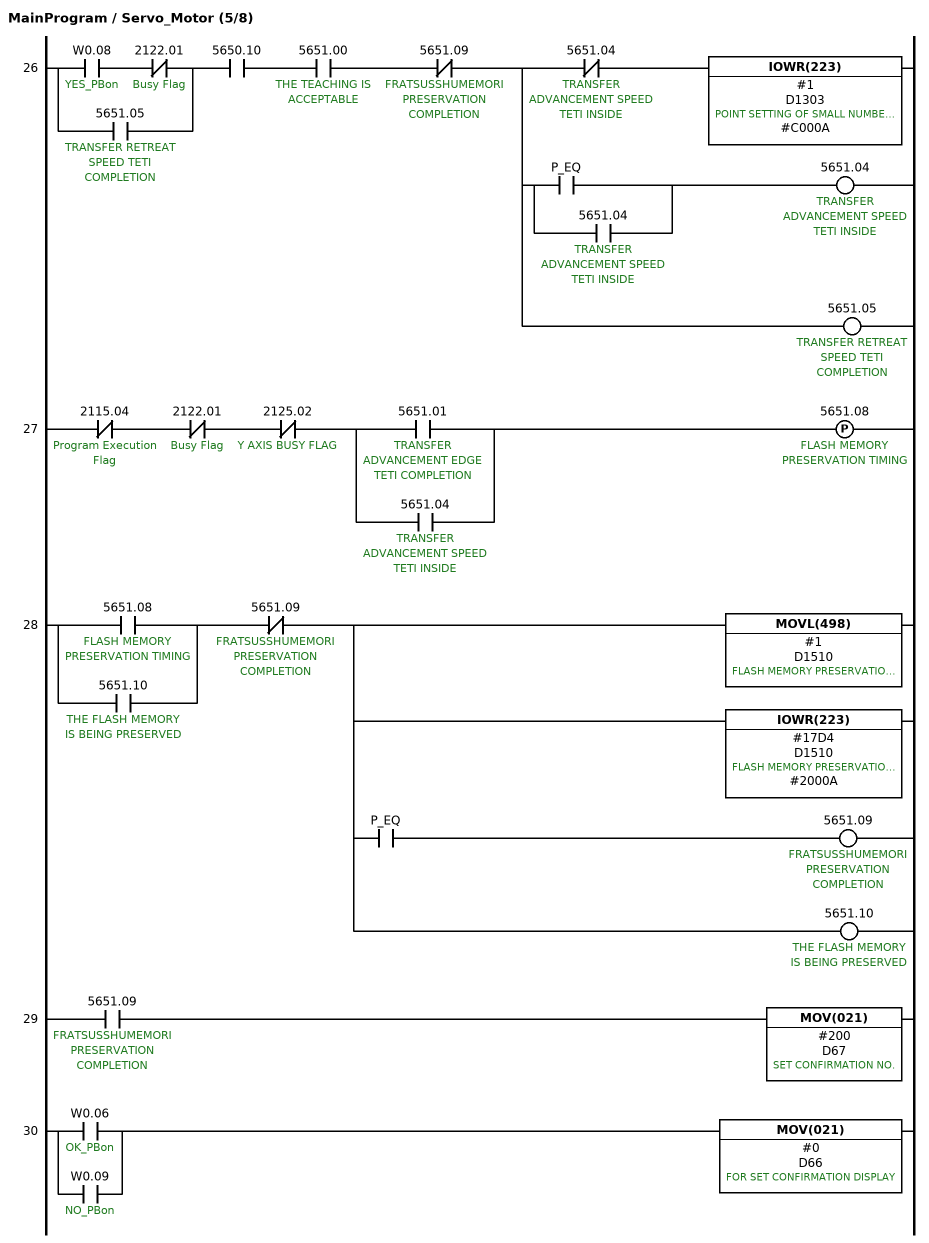
; [picture p216: MainProgram / Servo_Motor, rungs 26-30]
; rung 26
LD W0.08  ; YES_PBon
ANDNOT 2122.01  ; Busy Flag
OR 5651.05  ; TRANSFER RETREAT SPEED TETI COMPLETION
AND 5650.10
AND 5651.00  ; THE TEACHING IS ACCEPTABLE
ANDNOT 5651.09  ; FRATSUSSHUMEMORI PRESERVATION COMPLETION
OUT TR0
ANDNOT 5651.04  ; TRANSFER ADVANCEMENT SPEED TETI INSIDE
IOWR(223) #1 D1303 #C000A  ; POINT SETTING OF SMALL NUMBER OF ADVANCEMENT EDGES
LD TR0
LD P_EQ
OR 5651.04  ; TRANSFER ADVANCEMENT SPEED TETI INSIDE
ANDLD
OUT 5651.04  ; TRANSFER ADVANCEMENT SPEED TETI INSIDE
LD TR0
OUT 5651.05  ; TRANSFER RETREAT SPEED TETI COMPLETION
; rung 27
LDNOT 2115.04  ; Program Execution Flag
ANDNOT 2122.01  ; Busy Flag
ANDNOT 2125.02  ; Y AXIS BUSY FLAG
LD 5651.01  ; TRANSFER ADVANCEMENT EDGE TETI COMPLETION
OR 5651.04  ; TRANSFER ADVANCEMENT SPEED TETI INSIDE
ANDLD
DIFU(013) 5651.08  ; FLASH MEMORY PRESERVATION TIMING
; rung 28
LD 5651.08  ; FLASH MEMORY PRESERVATION TIMING
OR 5651.10  ; THE FLASH MEMORY IS BEING PRESERVED
ANDNOT 5651.09  ; FRATSUSSHUMEMORI PRESERVATION COMPLETION
OUT TR0
MOVL(498) #1 D1510  ; FLASH MEMORY PRESERVATION COMMAND
IOWR(223) #17D4 D1510 #2000A  ; FLASH MEMORY PRESERVATION COMMAND
AND P_EQ
OUT 5651.09  ; FRATSUSSHUMEMORI PRESERVATION COMPLETION
LD TR0
OUT 5651.10  ; THE FLASH MEMORY IS BEING PRESERVED
; rung 29
LD 5651.09  ; FRATSUSSHUMEMORI PRESERVATION COMPLETION
MOV(021) #200 D67  ; SET CONFIRMATION NO.
; rung 30
LD W0.06  ; OK_PBon
OR W0.09  ; NO_PBon
MOV(021) #0 D66  ; FOR SET CONFIRMATION DISPLAY

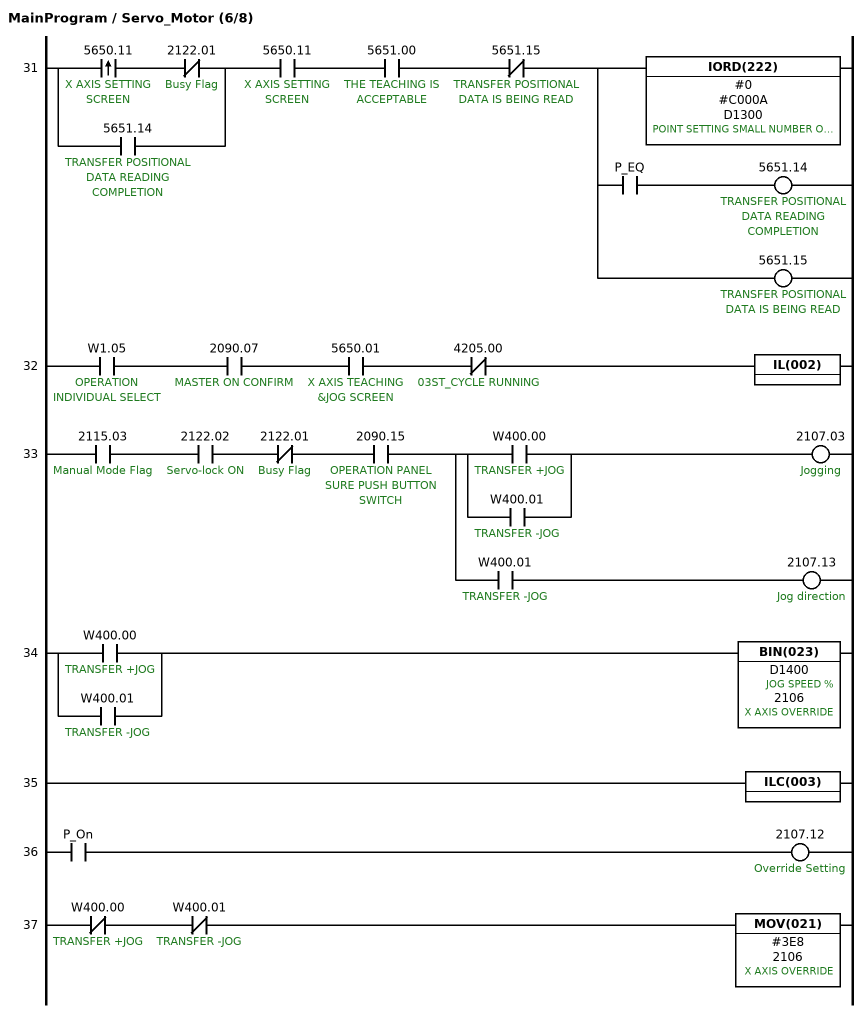
; rung 31
@LD 5650.11  ; X AXIS SETTING SCREEN
ANDNOT 2122.01  ; Busy Flag
OR 5651.14  ; TRANSFER POSITIONAL DATA READING COMPLETION
AND 5650.11  ; X AXIS SETTING SCREEN
AND 5651.00  ; THE TEACHING IS ACCEPTABLE
ANDNOT 5651.15  ; TRANSFER POSITIONAL DATA IS BEING READ
OUT TR0
IORD(222) #0 #C000A D1300  ; POINT SETTING SMALL NUMBER OF FORWARD SPEEDS
AND P_EQ
OUT 5651.14  ; TRANSFER POSITIONAL DATA READING COMPLETION
LD TR0
OUT 5651.15  ; TRANSFER POSITIONAL DATA IS BEING READ
; rung 32
LD W1.05  ; OPERATION INDIVIDUAL SELECT
AND 2090.07  ; MASTER ON CONFIRM
AND 5650.01  ; X AXIS TEACHING &JOG SCREEN
ANDNOT 4205.00  ; 03ST_CYCLE RUNNING
IL(002)
; rung 33
LD 2115.03  ; Manual Mode Flag
AND 2122.02  ; Servo-lock ON
ANDNOT 2122.01  ; Busy Flag
AND 2090.15  ; OPERATION PANEL SURE PUSH BUTTON SWITCH
OUT TR0
LD W400.00  ; TRANSFER +JOG
OR W400.01  ; TRANSFER -JOG
ANDLD
OUT 2107.03  ; Jogging
LD TR0
AND W400.01  ; TRANSFER -JOG
OUT 2107.13  ; Jog direction
; rung 34
LD W400.00  ; TRANSFER +JOG
OR W400.01  ; TRANSFER -JOG
BIN(023) D1400 2106  ; JOG SPEED %, X AXIS OVERRIDE
; rung 35
ILC(003)
; rung 36
LD P_On
OUT 2107.12  ; Override Setting
; rung 37
LDNOT W400.00  ; TRANSFER +JOG
ANDNOT W400.01  ; TRANSFER -JOG
MOV(021) #3E8 2106  ; X AXIS OVERRIDE

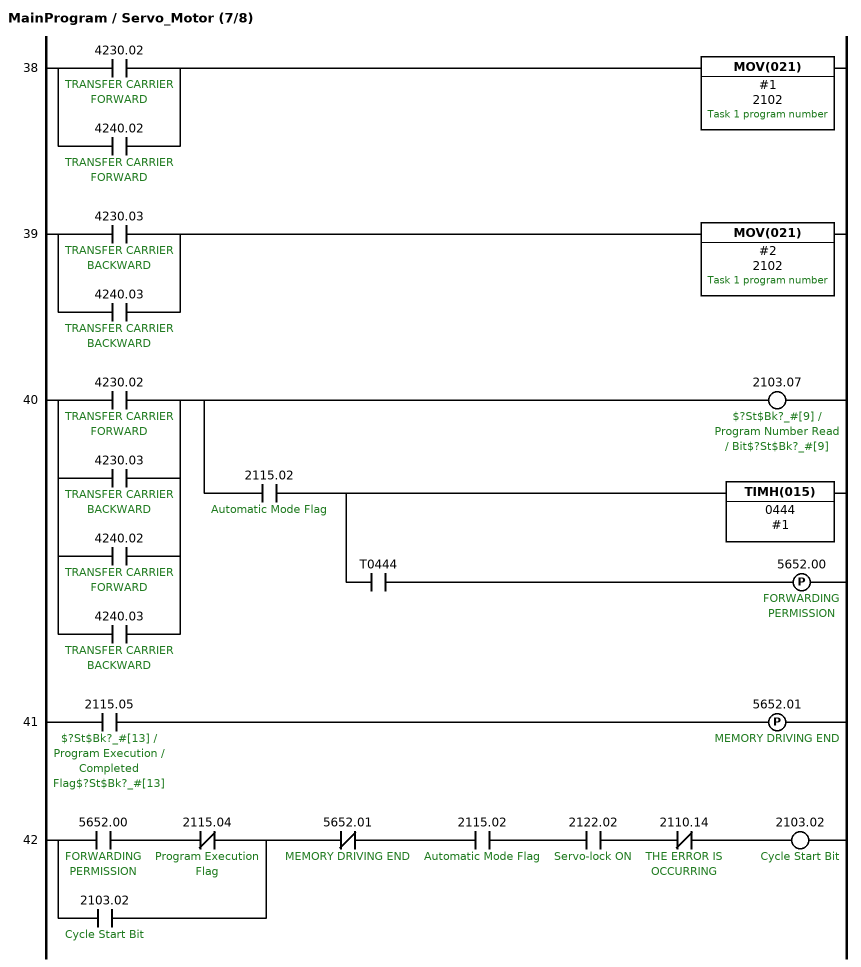
; rung 38
LD 4230.02  ; TRANSFER CARRIER FORWARD
OR 4240.02  ; TRANSFER CARRIER FORWARD
MOV(021) #1 2102  ; Task 1 program number
; rung 39
LD 4230.03  ; TRANSFER CARRIER BACKWARD
OR 4240.03  ; TRANSFER CARRIER BACKWARD
MOV(021) #2 2102  ; Task 1 program number
; rung 40
LD 4230.02  ; TRANSFER CARRIER FORWARD
OR 4230.03  ; TRANSFER CARRIER BACKWARD
OR 4240.02  ; TRANSFER CARRIER FORWARD
OR 4240.03  ; TRANSFER CARRIER BACKWARD
OUT 2103.07  ; $?St$Bk?_#[9] / Program Number Read / Bit$?St$Bk?_#[9]
AND 2115.02  ; Automatic Mode Flag
TIMH(015) 0444 #1
AND T0444
DIFU(013) 5652.00  ; FORWARDING PERMISSION
; rung 41
LD 2115.05  ; $?St$Bk?_#[13] / Program Execution / Completed Flag$?St$Bk?_#[13]
DIFU(013) 5652.01  ; MEMORY DRIVING END
; rung 42
LD 5652.00  ; FORWARDING PERMISSION
ANDNOT 2115.04  ; Program Execution Flag
OR 2103.02  ; Cycle Start Bit
ANDNOT 5652.01  ; MEMORY DRIVING END
AND 2115.02  ; Automatic Mode Flag
AND 2122.02  ; Servo-lock ON
ANDNOT 2110.14  ; THE ERROR IS OCCURRING
OUT 2103.02  ; Cycle Start Bit

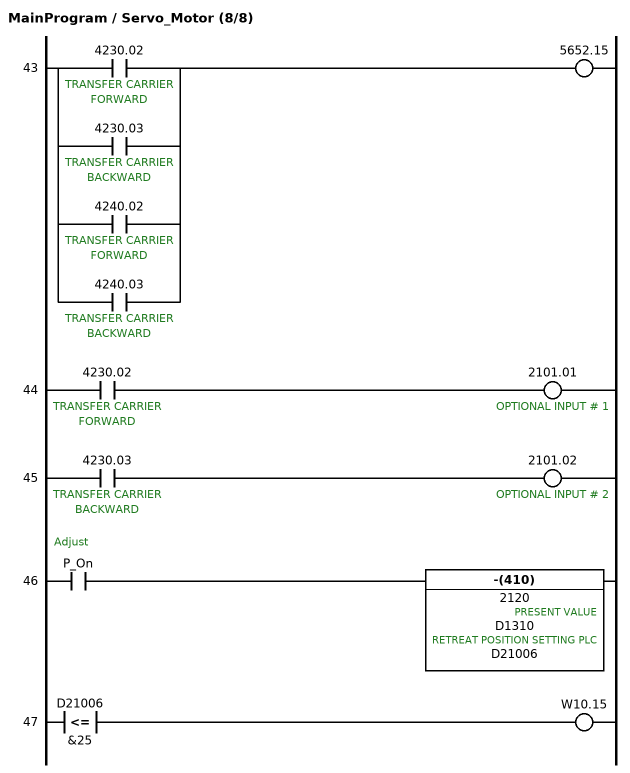
; rung 43
LD 4230.02  ; TRANSFER CARRIER FORWARD
OR 4230.03  ; TRANSFER CARRIER BACKWARD
OR 4240.02  ; TRANSFER CARRIER FORWARD
OR 4240.03  ; TRANSFER CARRIER BACKWARD
OUT 5652.15
; rung 44
LD 4230.02  ; TRANSFER CARRIER FORWARD
OUT 2101.01  ; OPTIONAL INPUT # 1
; rung 45
LD 4230.03  ; TRANSFER CARRIER BACKWARD
OUT 2101.02  ; OPTIONAL INPUT # 2
; rung 46: Adjust
LD P_On
-(410) 2120 D1310 D21006  ; PRESENT VALUE, RETREAT POSITION SETTING PLC
; rung 47
LD<=(315) D21006 &25
OUT W10.15

### Section BEARING_SUPPLY_LOADER

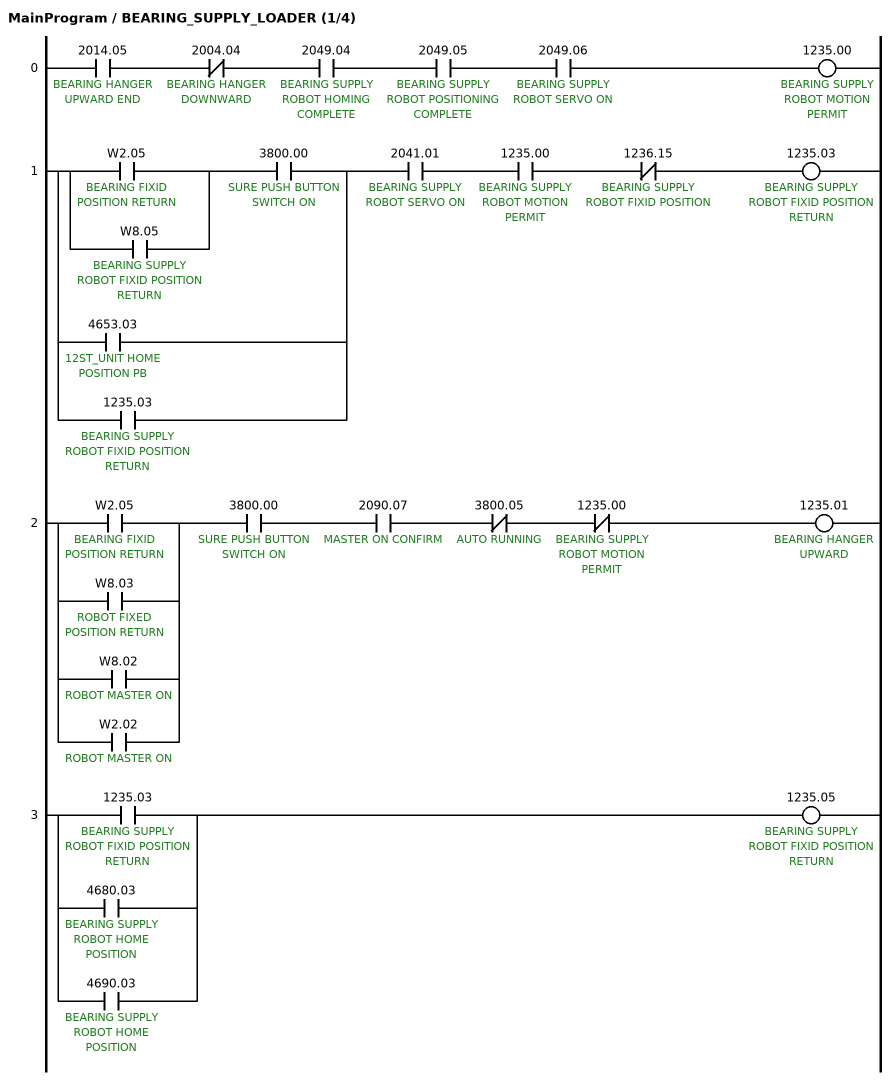
; rung 0
LD 2014.05  ; BEARING HANGER UPWARD END
ANDNOT 2004.04  ; BEARING HANGER DOWNWARD
AND 2049.04  ; BEARING SUPPLY ROBOT HOMING COMPLETE
AND 2049.05  ; BEARING SUPPLY ROBOT POSITIONING COMPLETE
AND 2049.06  ; BEARING SUPPLY ROBOT SERVO ON
OUT 1235.00  ; BEARING SUPPLY ROBOT MOTION PERMIT
; rung 1
LD W2.05  ; BEARING FIXID POSITION RETURN
OR W8.05  ; BEARING SUPPLY ROBOT FIXID POSITION RETURN
AND 3800.00  ; SURE PUSH BUTTON SWITCH ON
OR 4653.03  ; 12ST_UNIT HOME POSITION PB
OR 1235.03  ; BEARING SUPPLY ROBOT FIXID POSITION RETURN
AND 2041.01  ; BEARING SUPPLY ROBOT SERVO ON
AND 1235.00  ; BEARING SUPPLY ROBOT MOTION PERMIT
ANDNOT 1236.15  ; BEARING SUPPLY ROBOT FIXID POSITION
OUT 1235.03  ; BEARING SUPPLY ROBOT FIXID POSITION RETURN
; rung 2
LD W2.05  ; BEARING FIXID POSITION RETURN
OR W8.03  ; ROBOT FIXED POSITION RETURN
OR W8.02  ; ROBOT MASTER ON
OR W2.02  ; ROBOT MASTER ON
AND 3800.00  ; SURE PUSH BUTTON SWITCH ON
AND 2090.07  ; MASTER ON CONFIRM
ANDNOT 3800.05  ; AUTO RUNNING
ANDNOT 1235.00  ; BEARING SUPPLY ROBOT MOTION PERMIT
OUT 1235.01  ; BEARING HANGER UPWARD
; rung 3
LD 1235.03  ; BEARING SUPPLY ROBOT FIXID POSITION RETURN
OR 4680.03  ; BEARING SUPPLY ROBOT HOME POSITION
OR 4690.03  ; BEARING SUPPLY ROBOT HOME POSITION
OUT 1235.05  ; BEARING SUPPLY ROBOT FIXID POSITION RETURN

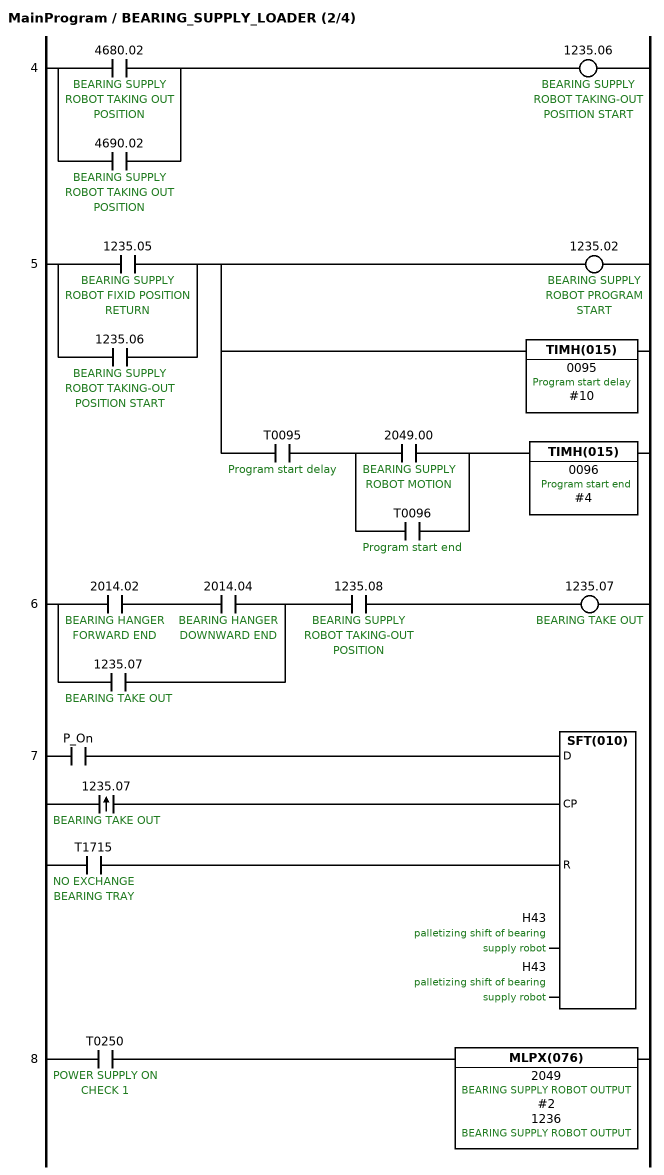
; rung 4
LD 4680.02  ; BEARING SUPPLY ROBOT TAKING OUT POSITION
OR 4690.02  ; BEARING SUPPLY ROBOT TAKING OUT POSITION
OUT 1235.06  ; BEARING SUPPLY ROBOT TAKING-OUT POSITION START
; rung 5
LD 1235.05  ; BEARING SUPPLY ROBOT FIXID POSITION RETURN
OR 1235.06  ; BEARING SUPPLY ROBOT TAKING-OUT POSITION START
OUT 1235.02  ; BEARING SUPPLY ROBOT PROGRAM START
TIMH(015) 0095 #10  ; Program start delay
AND T0095  ; Program start delay
LD 2049.00  ; BEARING SUPPLY ROBOT MOTION
OR T0096  ; Program start end
ANDLD
TIMH(015) 0096 #4  ; Program start end
; rung 6
LD 2014.02  ; BEARING HANGER FORWARD END
AND 2014.04  ; BEARING HANGER DOWNWARD END
OR 1235.07  ; BEARING TAKE OUT
AND 1235.08  ; BEARING SUPPLY ROBOT TAKING-OUT POSITION
OUT 1235.07  ; BEARING TAKE OUT
; rung 7
LD P_On
@LD 1235.07  ; BEARING TAKE OUT
LD T1715  ; NO EXCHANGE BEARING TRAY
SFT(010) H43 H43  ; palletizing shift of bearing supply robot
; rung 8
LD T0250  ; POWER SUPPLY ON CHECK 1
MLPX(076) 2049 #2 1236  ; BEARING SUPPLY ROBOT OUTPUT

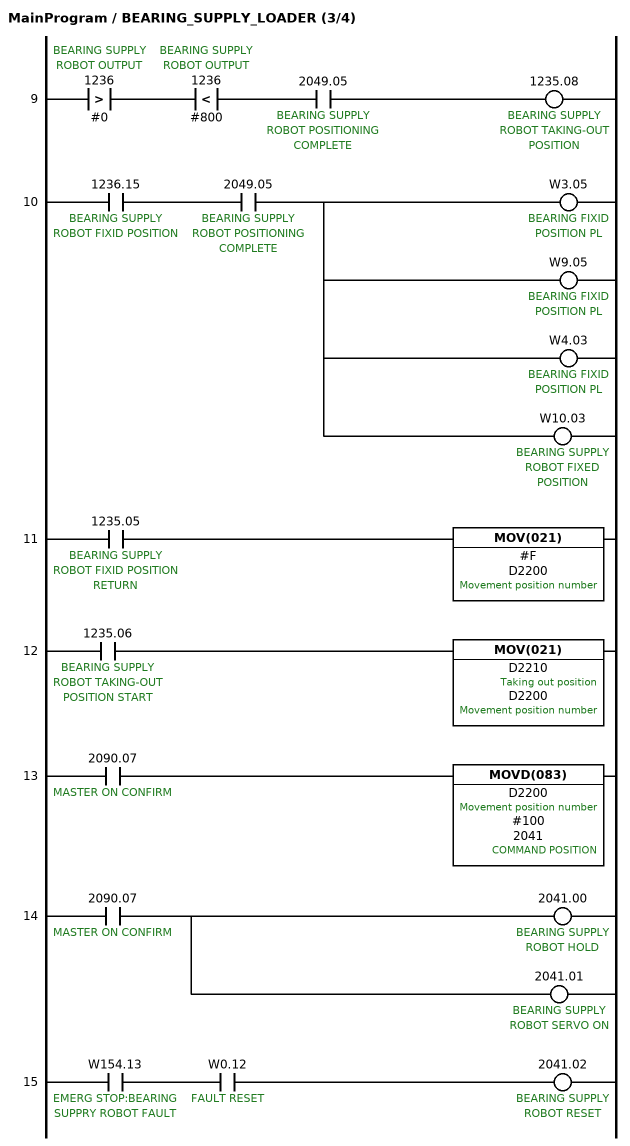
; rung 9
LD>(320) 1236 #0  ; BEARING SUPPLY ROBOT OUTPUT
AND<(310) 1236 #800  ; BEARING SUPPLY ROBOT OUTPUT
AND 2049.05  ; BEARING SUPPLY ROBOT POSITIONING COMPLETE
OUT 1235.08  ; BEARING SUPPLY ROBOT TAKING-OUT POSITION
; rung 10
LD 1236.15  ; BEARING SUPPLY ROBOT FIXID POSITION
AND 2049.05  ; BEARING SUPPLY ROBOT POSITIONING COMPLETE
OUT W3.05  ; BEARING FIXID POSITION PL
OUT W9.05  ; BEARING FIXID POSITION PL
OUT W4.03  ; BEARING FIXID POSITION PL
OUT W10.03  ; BEARING SUPPLY ROBOT FIXED POSITION
; rung 11
LD 1235.05  ; BEARING SUPPLY ROBOT FIXID POSITION RETURN
MOV(021) #F D2200  ; Movement position number
; rung 12
LD 1235.06  ; BEARING SUPPLY ROBOT TAKING-OUT POSITION START
MOV(021) D2210 D2200  ; Taking out position, Movement position number
; rung 13
LD 2090.07  ; MASTER ON CONFIRM
MOVD(083) D2200 #100 2041  ; Movement position number, COMMAND POSITION
; rung 14
LD 2090.07  ; MASTER ON CONFIRM
OUT 2041.00  ; BEARING SUPPLY ROBOT HOLD
OUT 2041.01  ; BEARING SUPPLY ROBOT SERVO ON
; rung 15
LD W154.13  ; EMERG STOP:BEARING SUPPRY ROBOT FAULT
AND W0.12  ; FAULT RESET
OUT 2041.02  ; BEARING SUPPLY ROBOT RESET

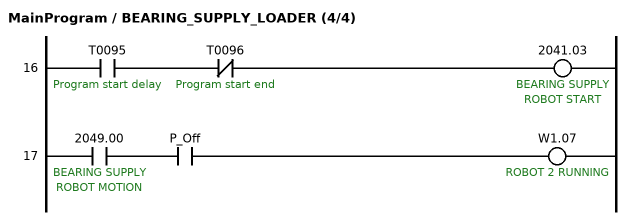
; rung 16
LD T0095  ; Program start delay
ANDNOT T0096  ; Program start end
OUT 2041.03  ; BEARING SUPPLY ROBOT START
; rung 17
LD 2049.00  ; BEARING SUPPLY ROBOT MOTION
AND P_Off
OUT W1.07  ; ROBOT 2 RUNNING

### Section SAVING_ENERGY_OF_FLURESCENT_LIGHT

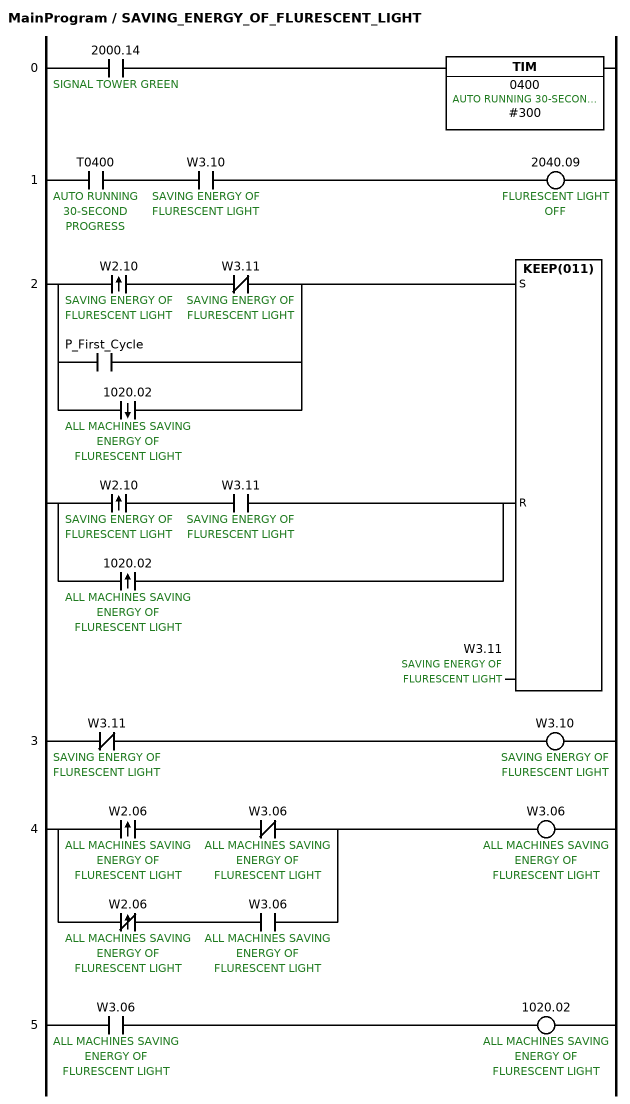
; rung 0
LD 2000.14  ; SIGNAL TOWER GREEN
TIM 0400 #300  ; AUTO RUNNING 30-SECOND PROGRESS
; rung 1
LD T0400  ; AUTO RUNNING 30-SECOND PROGRESS
AND W3.10  ; SAVING ENERGY OF FLURESCENT LIGHT
OUT 2040.09  ; FLURESCENT LIGHT OFF
; rung 2
@LD W2.10  ; SAVING ENERGY OF FLURESCENT LIGHT
ANDNOT W3.11  ; SAVING ENERGY OF FLURESCENT LIGHT
OR P_First_Cycle
%OR 1020.02  ; ALL MACHINES SAVING ENERGY OF FLURESCENT LIGHT
@LD W2.10  ; SAVING ENERGY OF FLURESCENT LIGHT
AND W3.11  ; SAVING ENERGY OF FLURESCENT LIGHT
@OR 1020.02  ; ALL MACHINES SAVING ENERGY OF FLURESCENT LIGHT
KEEP(011) W3.11  ; SAVING ENERGY OF FLURESCENT LIGHT
; rung 3
LDNOT W3.11  ; SAVING ENERGY OF FLURESCENT LIGHT
OUT W3.10  ; SAVING ENERGY OF FLURESCENT LIGHT
; rung 4
@LD W2.06  ; ALL MACHINES SAVING ENERGY OF FLURESCENT LIGHT
ANDNOT W3.06  ; ALL MACHINES SAVING ENERGY OF FLURESCENT LIGHT
@LDNOT W2.06  ; ALL MACHINES SAVING ENERGY OF FLURESCENT LIGHT
AND W3.06  ; ALL MACHINES SAVING ENERGY OF FLURESCENT LIGHT
ORLD
OUT W3.06  ; ALL MACHINES SAVING ENERGY OF FLURESCENT LIGHT
; rung 5
LD W3.06  ; ALL MACHINES SAVING ENERGY OF FLURESCENT LIGHT
OUT 1020.02  ; ALL MACHINES SAVING ENERGY OF FLURESCENT LIGHT

### Section CYCLE_TIME

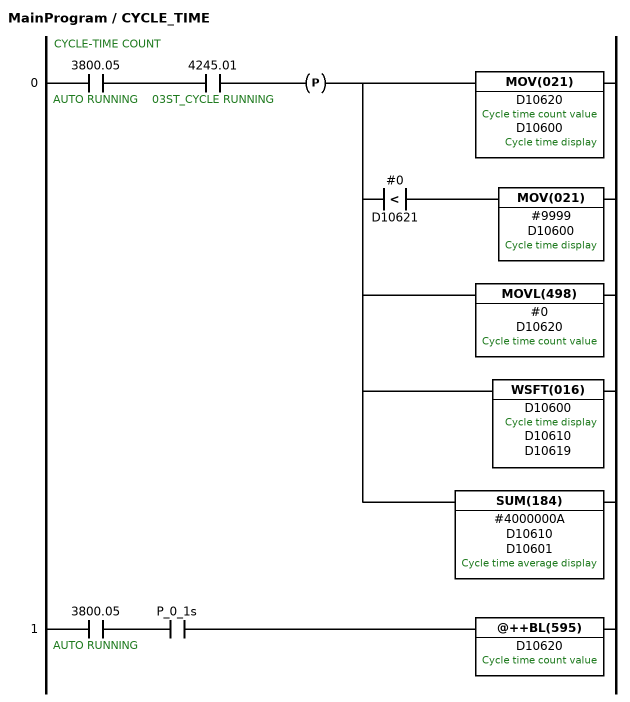
; rung 0: CYCLE-TIME COUNT
LD 3800.05  ; AUTO RUNNING
AND 4245.01  ; 03ST_CYCLE RUNNING
UP(521)
OUT TR0
MOV(021) D10620 D10600  ; Cycle time count value, Cycle time display
AND<(310) #0 D10621
MOV(021) #9999 D10600  ; Cycle time display
LD TR0
MOVL(498) #0 D10620  ; Cycle time count value
WSFT(016) D10600 D10610 D10619  ; Cycle time display
SUM(184) #4000000A D10610 D10601  ; Cycle time average display
; rung 1
LD 3800.05  ; AUTO RUNNING
AND P_0_1s
@++BL(595) D10620  ; Cycle time count value

### Section PRODUCTION_SITUATION

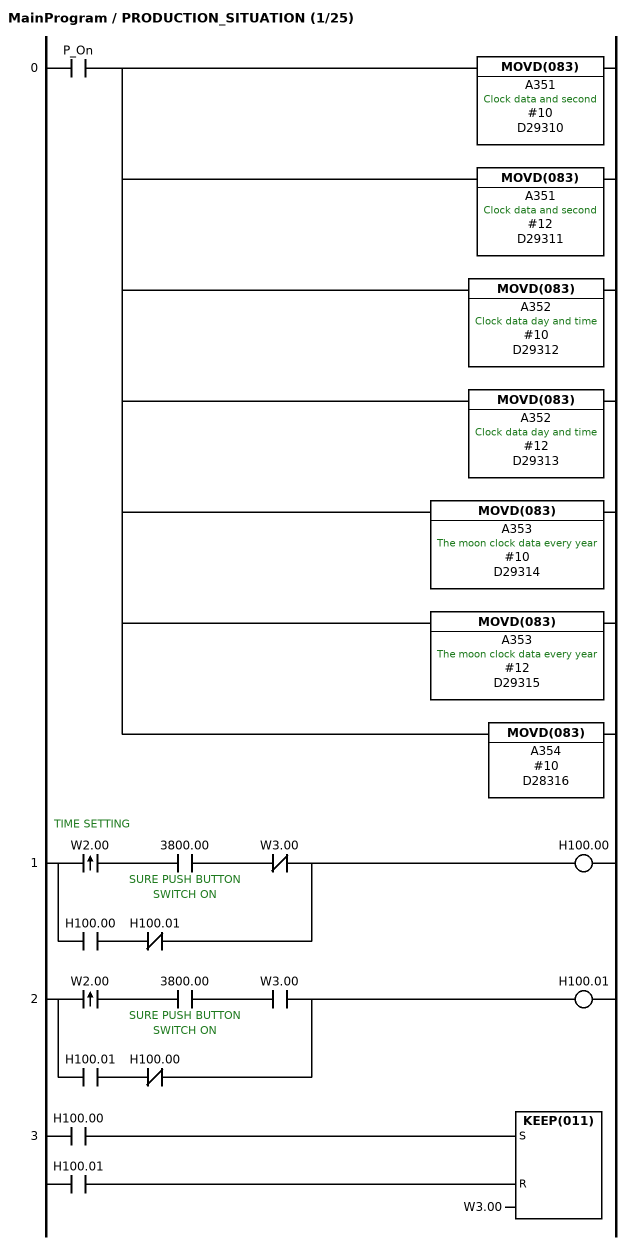
; rung 0
LD P_On
MOVD(083) A351 #10 D29310  ; Clock data and second
MOVD(083) A351 #12 D29311  ; Clock data and second
MOVD(083) A352 #10 D29312  ; Clock data day and time
MOVD(083) A352 #12 D29313  ; Clock data day and time
MOVD(083) A353 #10 D29314  ; The moon clock data every year
MOVD(083) A353 #12 D29315  ; The moon clock data every year
MOVD(083) A354 #10 D28316
; rung 1: TIME SETTING
@LD W2.00
AND 3800.00  ; SURE PUSH BUTTON SWITCH ON
ANDNOT W3.00
LD H100.00
ANDNOT H100.01
ORLD
OUT H100.00
; rung 2
@LD W2.00
AND 3800.00  ; SURE PUSH BUTTON SWITCH ON
AND W3.00
LD H100.01
ANDNOT H100.00
ORLD
OUT H100.01
; rung 3
LD H100.00
LD H100.01
KEEP(011) W3.00

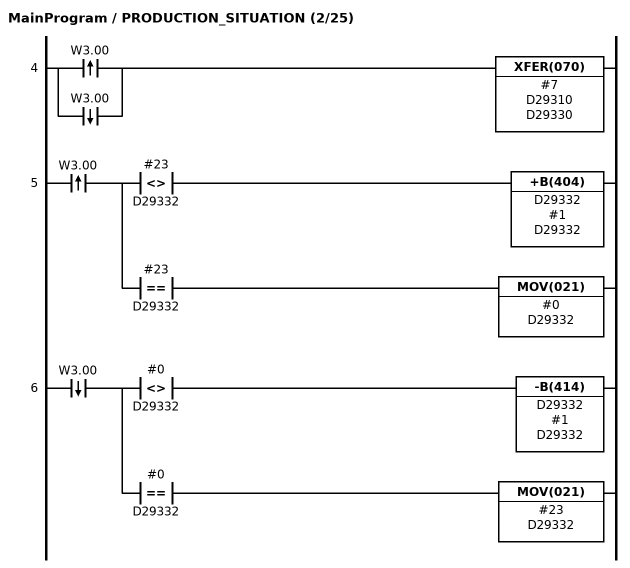
; rung 4
@LD W3.00
%OR W3.00
XFER(070) #7 D29310 D29330
; rung 5
@LD W3.00
OUT TR0
AND<>(305) #23 D29332
+B(404) D29332 #1 D29332
LD TR0
AND=(300) #23 D29332
MOV(021) #0 D29332
; rung 6
%LD W3.00
OUT TR0
AND<>(305) #0 D29332
-B(414) D29332 #1 D29332
LD TR0
AND=(300) #0 D29332
MOV(021) #23 D29332

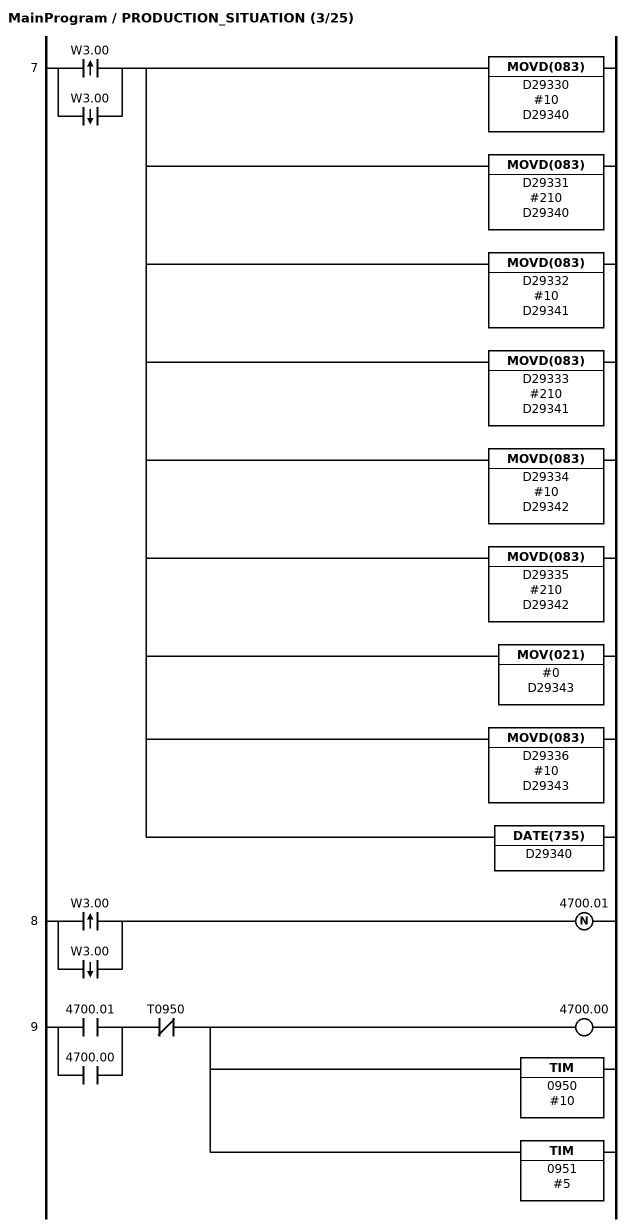
; rung 7
@LD W3.00
%OR W3.00
MOVD(083) D29330 #10 D29340
MOVD(083) D29331 #210 D29340
MOVD(083) D29332 #10 D29341
MOVD(083) D29333 #210 D29341
MOVD(083) D29334 #10 D29342
MOVD(083) D29335 #210 D29342
MOV(021) #0 D29343
MOVD(083) D29336 #10 D29343
DATE(735) D29340
; rung 8
@LD W3.00
%OR W3.00
DIFD(014) 4700.01
; rung 9
LD 4700.01
OR 4700.00
ANDNOT T0950
OUT 4700.00
TIM 0950 #10
TIM 0951 #5

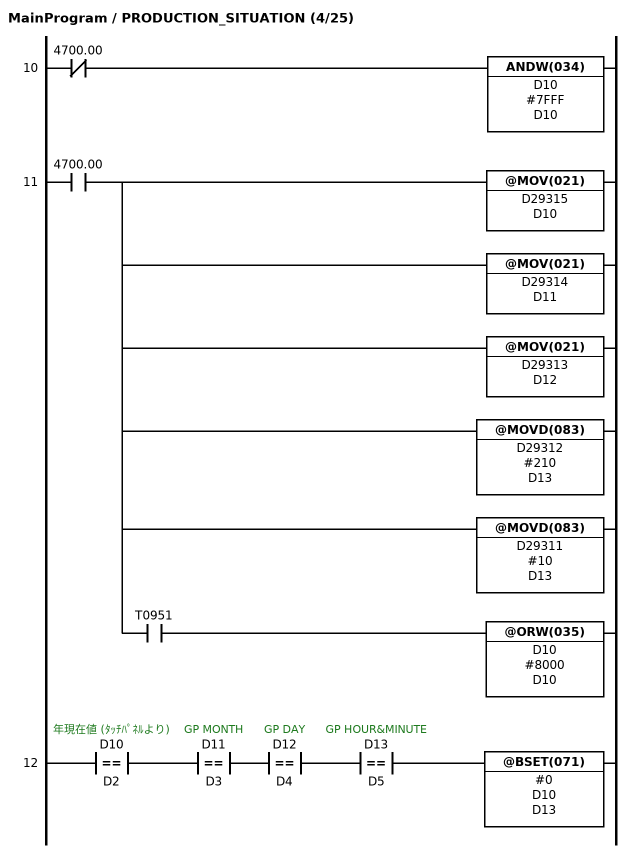
; rung 10
LDNOT 4700.00
ANDW(034) D10 #7FFF D10
; rung 11
LD 4700.00
@MOV(021) D29315 D10
@MOV(021) D29314 D11
@MOV(021) D29313 D12
@MOVD(083) D29312 #210 D13
@MOVD(083) D29311 #10 D13
AND T0951
@ORW(035) D10 #8000 D10
; rung 12
LD=(300) D10 D2  ; 年現在値 (ﾀｯﾁﾊﾟﾈﾙより)
AND=(300) D11 D3  ; GP MONTH
AND=(300) D12 D4  ; GP DAY
AND=(300) D13 D5  ; GP HOUR&MINUTE
@BSET(071) #0 D10 D13

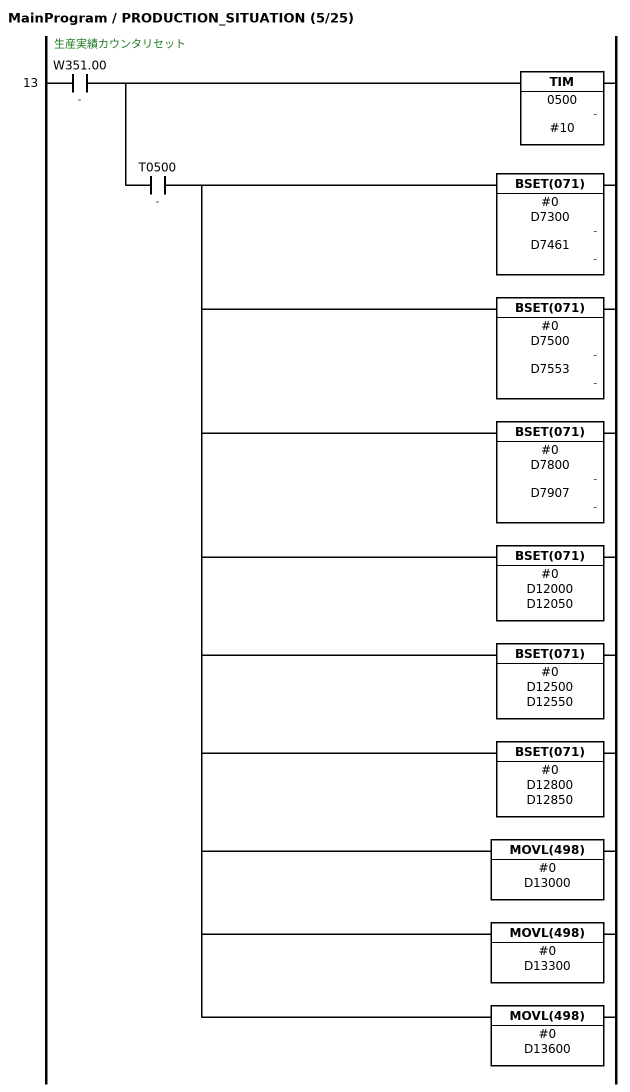
; rung 13: 生産実績カウンタリセット
LD W351.00  ; -
TIM 0500 #10  ; -
AND T0500  ; -
BSET(071) #0 D7300 D7461  ; -
BSET(071) #0 D7500 D7553  ; -
BSET(071) #0 D7800 D7907  ; -
BSET(071) #0 D12000 D12050
BSET(071) #0 D12500 D12550
BSET(071) #0 D12800 D12850
MOVL(498) #0 D13000
MOVL(498) #0 D13300
MOVL(498) #0 D13600

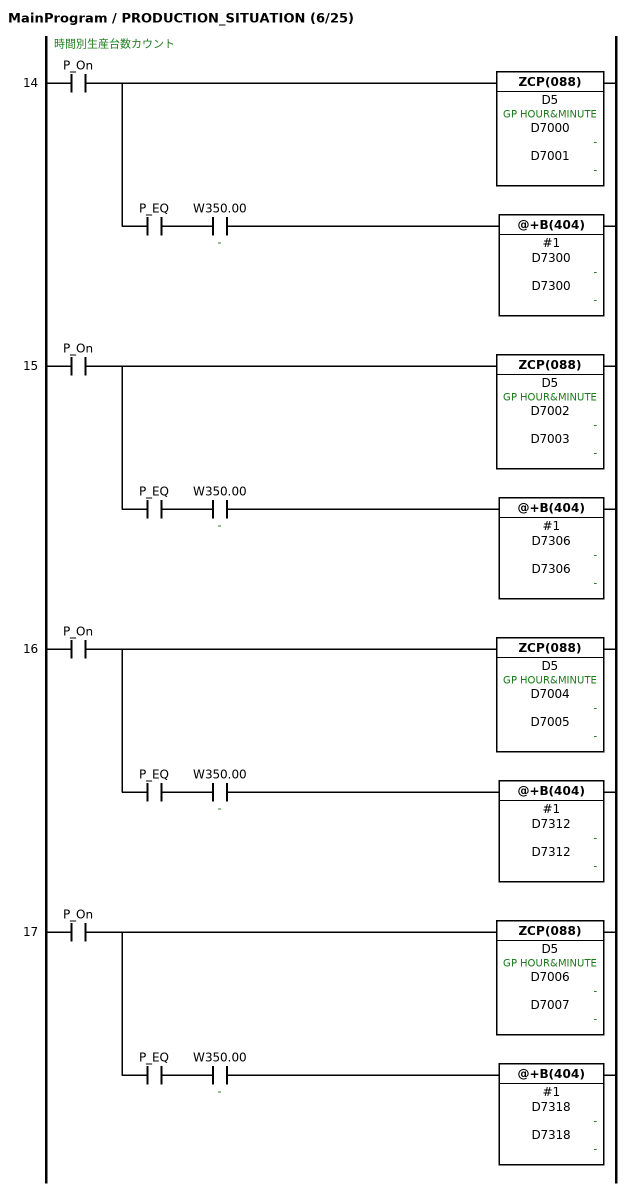
; rung 14: 時間別生産台数カウント
LD P_On
ZCP(088) D5 D7000 D7001  ; GP HOUR&MINUTE, -
AND P_EQ
AND W350.00  ; -
@+B(404) #1 D7300 D7300  ; -
; rung 15
LD P_On
ZCP(088) D5 D7002 D7003  ; GP HOUR&MINUTE, -
AND P_EQ
AND W350.00  ; -
@+B(404) #1 D7306 D7306  ; -
; rung 16
LD P_On
ZCP(088) D5 D7004 D7005  ; GP HOUR&MINUTE, -
AND P_EQ
AND W350.00  ; -
@+B(404) #1 D7312 D7312  ; -
; rung 17
LD P_On
ZCP(088) D5 D7006 D7007  ; GP HOUR&MINUTE, -
AND P_EQ
AND W350.00  ; -
@+B(404) #1 D7318 D7318  ; -

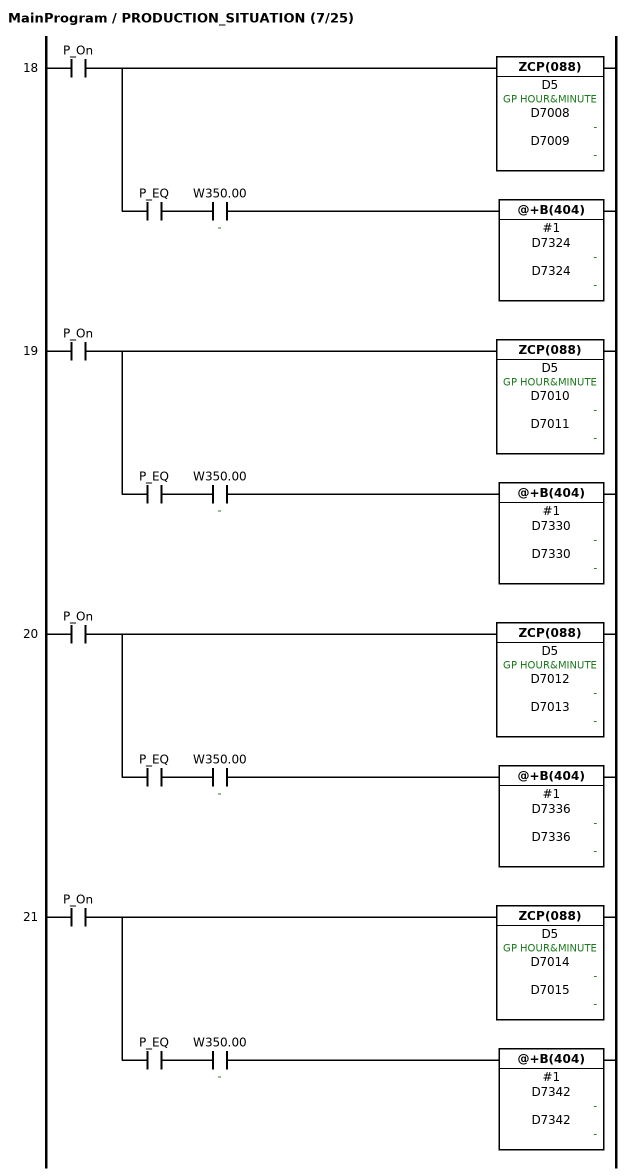
; rung 18
LD P_On
ZCP(088) D5 D7008 D7009  ; GP HOUR&MINUTE, -
AND P_EQ
AND W350.00  ; -
@+B(404) #1 D7324 D7324  ; -
; rung 19
LD P_On
ZCP(088) D5 D7010 D7011  ; GP HOUR&MINUTE, -
AND P_EQ
AND W350.00  ; -
@+B(404) #1 D7330 D7330  ; -
; rung 20
LD P_On
ZCP(088) D5 D7012 D7013  ; GP HOUR&MINUTE, -
AND P_EQ
AND W350.00  ; -
@+B(404) #1 D7336 D7336  ; -
; rung 21
LD P_On
ZCP(088) D5 D7014 D7015  ; GP HOUR&MINUTE, -
AND P_EQ
AND W350.00  ; -
@+B(404) #1 D7342 D7342  ; -

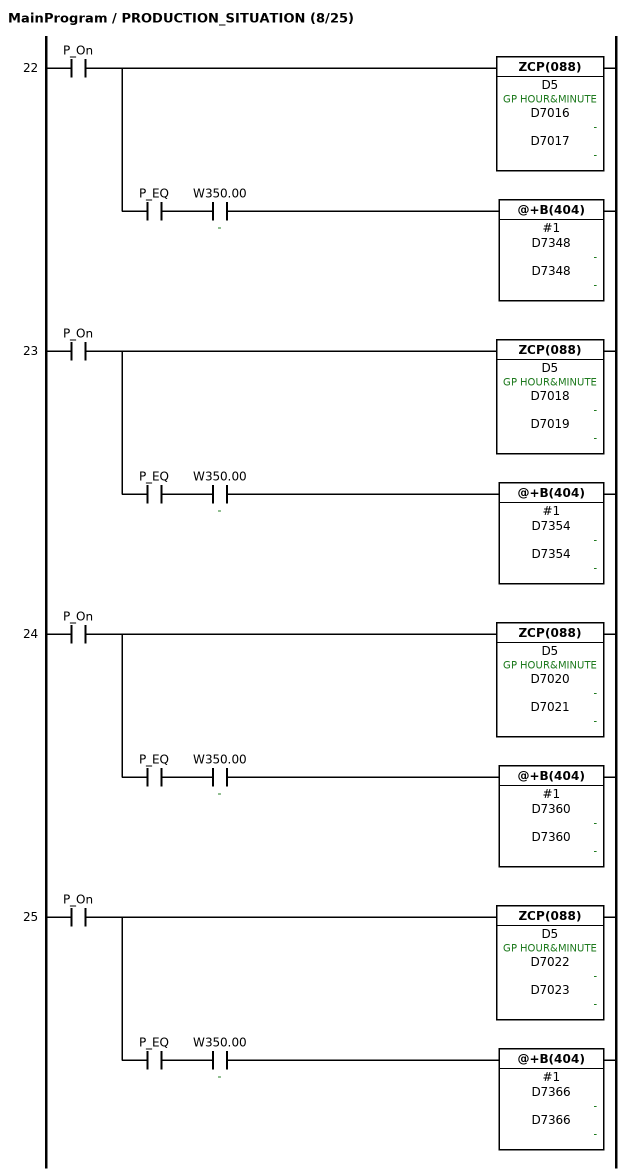
; rung 22
LD P_On
ZCP(088) D5 D7016 D7017  ; GP HOUR&MINUTE, -
AND P_EQ
AND W350.00  ; -
@+B(404) #1 D7348 D7348  ; -
; rung 23
LD P_On
ZCP(088) D5 D7018 D7019  ; GP HOUR&MINUTE, -
AND P_EQ
AND W350.00  ; -
@+B(404) #1 D7354 D7354  ; -
; rung 24
LD P_On
ZCP(088) D5 D7020 D7021  ; GP HOUR&MINUTE, -
AND P_EQ
AND W350.00  ; -
@+B(404) #1 D7360 D7360  ; -
; rung 25
LD P_On
ZCP(088) D5 D7022 D7023  ; GP HOUR&MINUTE, -
AND P_EQ
AND W350.00  ; -
@+B(404) #1 D7366 D7366  ; -

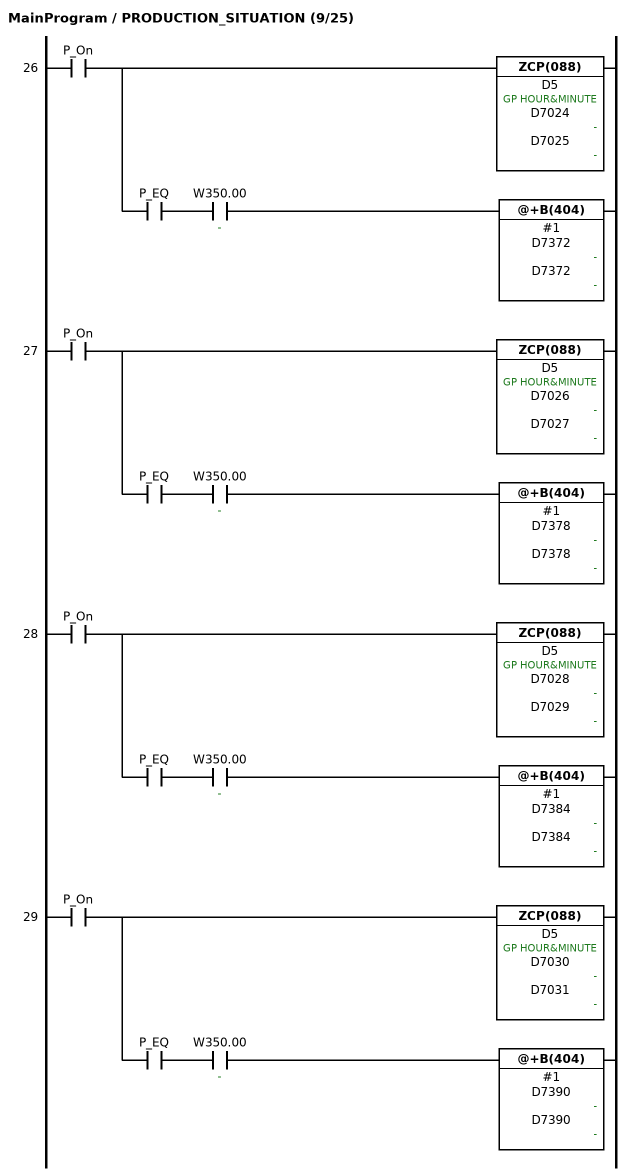
; rung 26
LD P_On
ZCP(088) D5 D7024 D7025  ; GP HOUR&MINUTE, -
AND P_EQ
AND W350.00  ; -
@+B(404) #1 D7372 D7372  ; -
; rung 27
LD P_On
ZCP(088) D5 D7026 D7027  ; GP HOUR&MINUTE, -
AND P_EQ
AND W350.00  ; -
@+B(404) #1 D7378 D7378  ; -
; rung 28
LD P_On
ZCP(088) D5 D7028 D7029  ; GP HOUR&MINUTE, -
AND P_EQ
AND W350.00  ; -
@+B(404) #1 D7384 D7384  ; -
; rung 29
LD P_On
ZCP(088) D5 D7030 D7031  ; GP HOUR&MINUTE, -
AND P_EQ
AND W350.00  ; -
@+B(404) #1 D7390 D7390  ; -

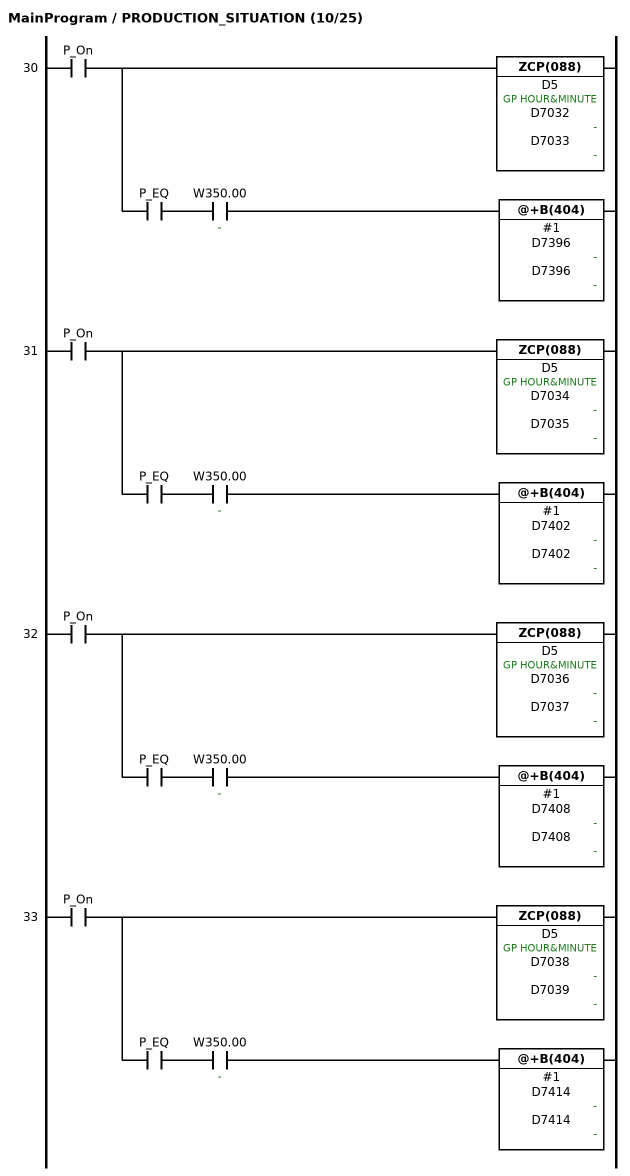
; rung 30
LD P_On
ZCP(088) D5 D7032 D7033  ; GP HOUR&MINUTE, -
AND P_EQ
AND W350.00  ; -
@+B(404) #1 D7396 D7396  ; -
; rung 31
LD P_On
ZCP(088) D5 D7034 D7035  ; GP HOUR&MINUTE, -
AND P_EQ
AND W350.00  ; -
@+B(404) #1 D7402 D7402  ; -
; rung 32
LD P_On
ZCP(088) D5 D7036 D7037  ; GP HOUR&MINUTE, -
AND P_EQ
AND W350.00  ; -
@+B(404) #1 D7408 D7408  ; -
; rung 33
LD P_On
ZCP(088) D5 D7038 D7039  ; GP HOUR&MINUTE, -
AND P_EQ
AND W350.00  ; -
@+B(404) #1 D7414 D7414  ; -

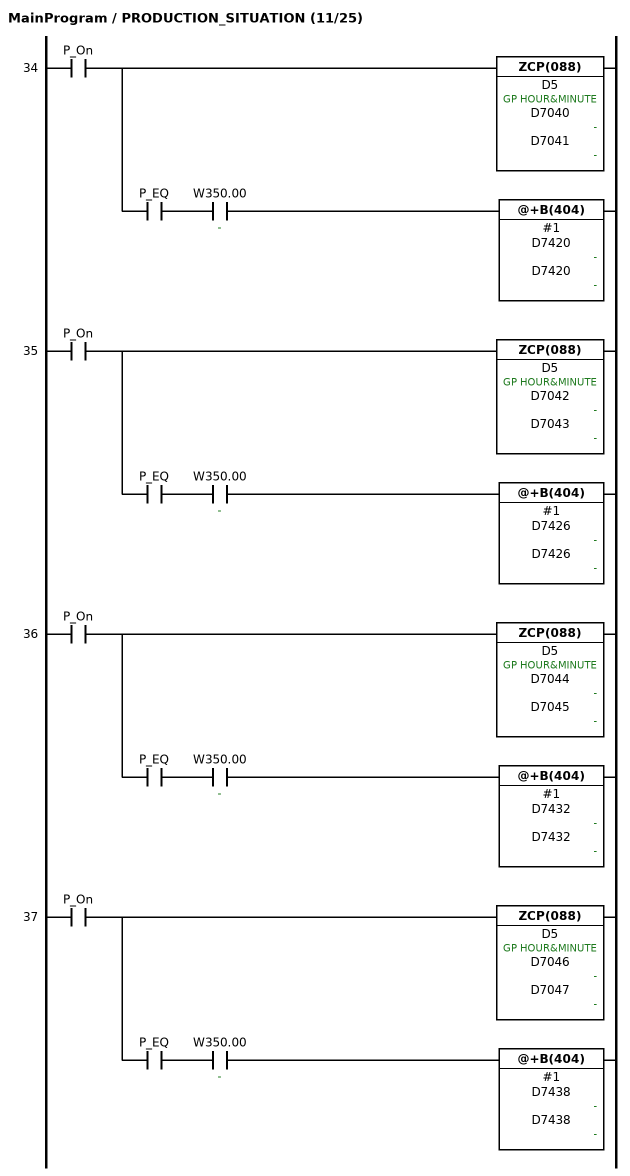
; rung 34
LD P_On
ZCP(088) D5 D7040 D7041  ; GP HOUR&MINUTE, -
AND P_EQ
AND W350.00  ; -
@+B(404) #1 D7420 D7420  ; -
; rung 35
LD P_On
ZCP(088) D5 D7042 D7043  ; GP HOUR&MINUTE, -
AND P_EQ
AND W350.00  ; -
@+B(404) #1 D7426 D7426  ; -
; rung 36
LD P_On
ZCP(088) D5 D7044 D7045  ; GP HOUR&MINUTE, -
AND P_EQ
AND W350.00  ; -
@+B(404) #1 D7432 D7432  ; -
; rung 37
LD P_On
ZCP(088) D5 D7046 D7047  ; GP HOUR&MINUTE, -
AND P_EQ
AND W350.00  ; -
@+B(404) #1 D7438 D7438  ; -

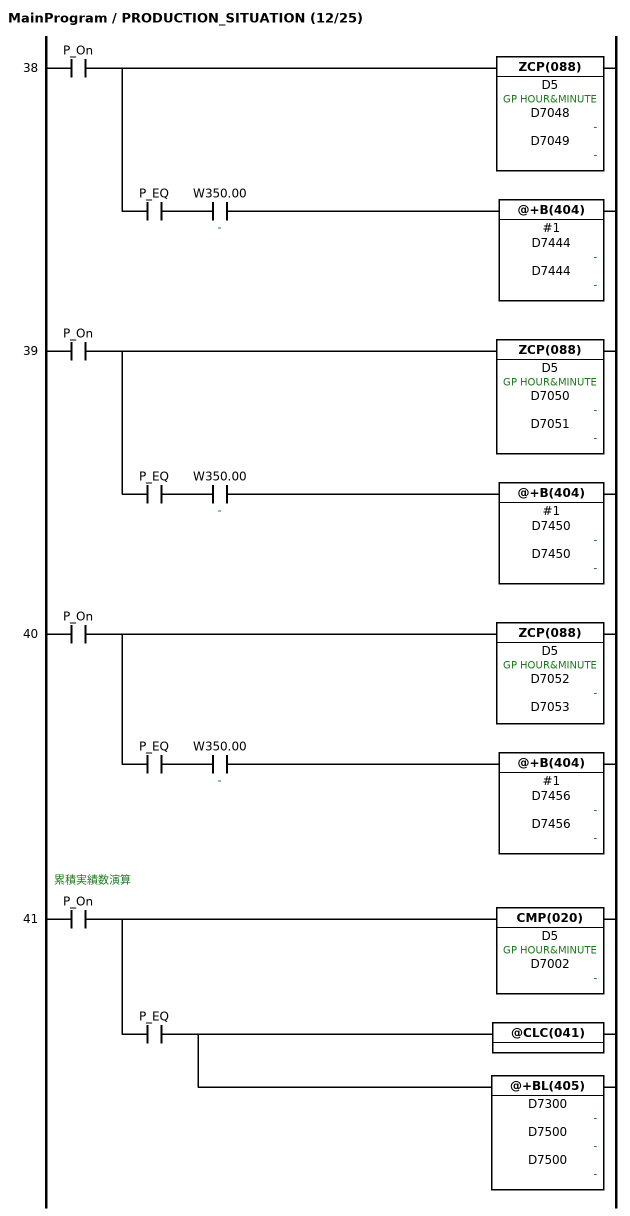
; rung 38
LD P_On
ZCP(088) D5 D7048 D7049  ; GP HOUR&MINUTE, -
AND P_EQ
AND W350.00  ; -
@+B(404) #1 D7444 D7444  ; -
; rung 39
LD P_On
ZCP(088) D5 D7050 D7051  ; GP HOUR&MINUTE, -
AND P_EQ
AND W350.00  ; -
@+B(404) #1 D7450 D7450  ; -
; rung 40
LD P_On
ZCP(088) D5 D7052 D7053  ; GP HOUR&MINUTE, -
AND P_EQ
AND W350.00  ; -
@+B(404) #1 D7456 D7456  ; -
; rung 41: 累積実績数演算
LD P_On
CMP(020) D5 D7002  ; GP HOUR&MINUTE, -
AND P_EQ
@CLC(041)
@+BL(405) D7300 D7500 D7500  ; -

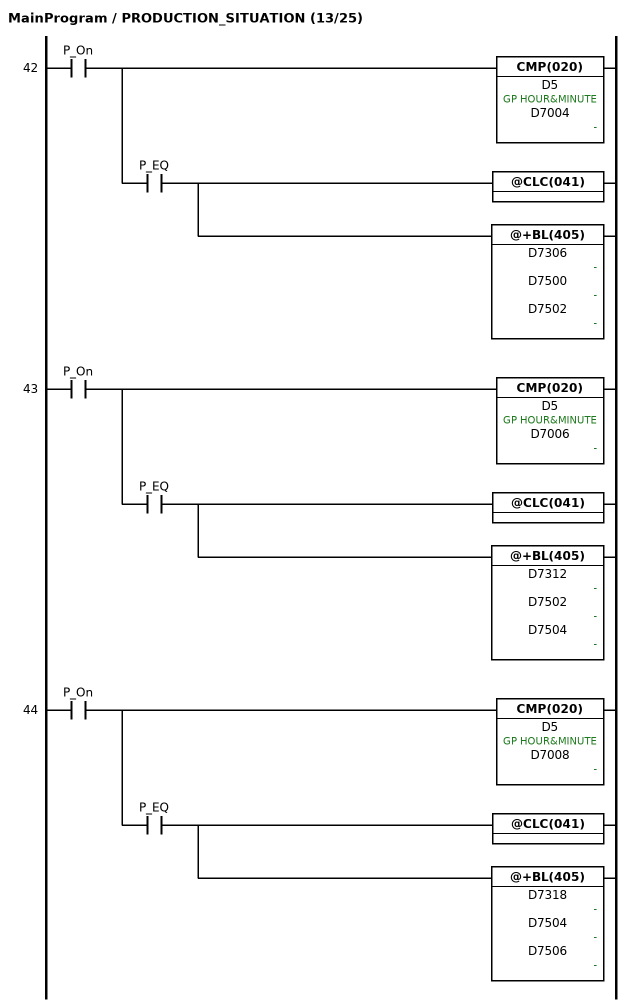
; rung 42
LD P_On
CMP(020) D5 D7004  ; GP HOUR&MINUTE, -
AND P_EQ
@CLC(041)
@+BL(405) D7306 D7500 D7502  ; -
; rung 43
LD P_On
CMP(020) D5 D7006  ; GP HOUR&MINUTE, -
AND P_EQ
@CLC(041)
@+BL(405) D7312 D7502 D7504  ; -
; rung 44
LD P_On
CMP(020) D5 D7008  ; GP HOUR&MINUTE, -
AND P_EQ
@CLC(041)
@+BL(405) D7318 D7504 D7506  ; -

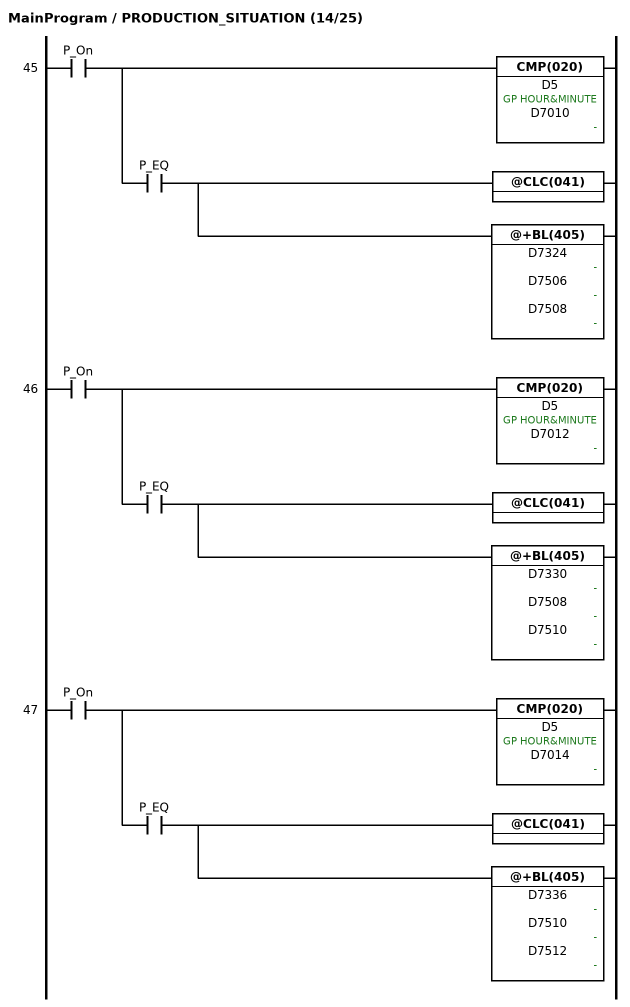
; rung 45
LD P_On
CMP(020) D5 D7010  ; GP HOUR&MINUTE, -
AND P_EQ
@CLC(041)
@+BL(405) D7324 D7506 D7508  ; -
; rung 46
LD P_On
CMP(020) D5 D7012  ; GP HOUR&MINUTE, -
AND P_EQ
@CLC(041)
@+BL(405) D7330 D7508 D7510  ; -
; rung 47
LD P_On
CMP(020) D5 D7014  ; GP HOUR&MINUTE, -
AND P_EQ
@CLC(041)
@+BL(405) D7336 D7510 D7512  ; -

